{attribute 'GeneratedUsingTerminal: APS1003-5000-0016'}
{attribute addProperty BoxType "APS1003-5000-0016"}
{attribute addProperty Id "FB_InputsAT %I*FB_Inputs_F0F03BDD308WcStateAT %I*WcState_9091E0EB2InfoDataAT %I*InfoData_A7436BC610"}
{attribute addProperty CRC "2761708599"}
{attribute addProperty Size "320"}
TYPE APS1003_A49C5437 :
STRUCT
	{attribute addProperty Name "FB_Inputs"}
	FB_Inputs : FB_Inputs_F0F03BDD;
	{attribute addProperty Name "WcState"}
	WcState : WcState_9091E0EB;
	{attribute addProperty Name "InfoData"}
	InfoData : InfoData_A7436BC6;
END_STRUCT
END_TYPE

(* stored: Version 1.2.0.0, ProductVersion 3.1.4024.9
   DUT APS1003_A49C5437: Id {a377d59a-75ca-48e9-857f-0da27706c399} *)
